// TIA Portal V20 export
DATA_BLOCK "Data_To_Safety"   // DB3
{ S7_Optimized_Access := 'TRUE' }
// stored: MemoryReserve 100
   VAR
      Reset_ESTOPS : Bool;
      Reset_REI : Bool;
      PLC_Hall4_Safety : Bool;
   END_VAR
BEGIN
END_DATA_BLOCK
